FUNCTION_BLOCK EcMasterConfDevices IMPLEMENTS IEcTask
VAR_INPUT
END_VAR
VAR_OUTPUT
END_VAR
VAR
	iState : INT;
	masterConfDevices : Tc2_EtherCAT.FB_EcGetConfSlaves;
	_confDevices : ARRAY[0..Tc2_EtherCAT.EC_MAX_SLAVES] OF Tc2_EtherCAT.ST_EcSlaveConfigData;
	_execute: BOOL;
	_done: BOOL;
	_busy: BOOL;	
	_error: BOOL;
	_netId: AMSNETID;
END_VAR

CASE iState OF
	0:
		IF _execute THEN
			_done := FALSE;
			_busy := TRUE;
			_error := FALSE;
			masterConfDevices.bExecute := TRUE;
			IF masterConfDevices.bBusy THEN
				iState := 10;
				_execute := FALSE;
			END_IF
		END_IF
	10:
		IF NOT masterConfDevices.bBusy THEN
			IF NOT masterConfDevices.bError THEN
				_done := TRUE;
			ELSE
				_error := TRUE;
			END_IF
			_busy := FALSE;
			masterConfDevices.bExecute := FALSE;
			iState := 0;
		END_IF
END_CASE

masterConfDevices(sNetId := Tc2_System.F_CreateAmsNetId(nIds := NetId), 
					pArrEcConfSlaveInfo := ADR(_confDevices), 
					cbBufLen := SIZEOF(_confDevices));

{warning 'add method implementation '}
METHOD Abort : BOOL
masterConfDevices.bExecute := FALSE;
_busy := FALSE;
_execute := FALSE;
Abort := TRUE;
iState := 0;
END_METHOD

{warning 'add property implementation'}
PROPERTY Busy : BOOL
GET
Busy := _busy;
END_GET
END_PROPERTY

PROPERTY ConfiguredDevices : reference to array[0..Ec_Max_slaves] of St_ecslaveconfigdata
GET
ConfiguredDevices REF= _confDevices;
END_GET
END_PROPERTY

{warning 'add property implementation'}
PROPERTY Done : BOOL
GET
Done := _done;
END_GET
END_PROPERTY

{warning 'add property implementation'}
PROPERTY Error : BOOL
GET
Error := _error;
END_GET
END_PROPERTY

{warning 'add method implementation '}
METHOD Execute : BOOL
IF NOT masterConfDevices.bBusy THEN
	Execute := _execute := true;
END_IF
END_METHOD

{warning 'add property implementation'}
PROPERTY NetID : amsnetid
GET
NetID := _netId;
END_GET
SET
_netId := NetID;
END_SET
END_PROPERTY

PROPERTY NumberConfDevices : udint
GET
NumberConfDevices := masterConfDevices.nSlaves;
END_GET
END_PROPERTY

END_FUNCTION_BLOCK

(* stored: Version 1.1.0.1, ProductVersion 3.1.4024.11
   POU EcMasterConfDevices: Id {db18c880-11a0-493e-8ecc-75b7bb7d5ee1}, SpecialFunc None
   Method Abort: Id {29f4c6c7-c295-4b3b-88e0-1affbc2a49a0}
   Property Busy: Id {fbdf4132-a177-46bc-967b-0566d7f33115}
   Get Get: Id {5d58dddb-706d-4e38-b676-e06487ff79db}
   Property ConfiguredDevices: Id {fb01f319-f3bb-49a5-aaac-41e3704dce79}
   Get Get: Id {9f6170b9-866e-4cce-be3c-72b47ca25254}
   Property Done: Id {b48d60e5-568a-4737-82f5-f064f1fec13f}
   Get Get: Id {98963513-5a99-4ba5-9e68-de084642d9dc}
   Property Error: Id {26c57861-0c4e-4191-bdd5-0866724eb110}
   Get Get: Id {e6fa895d-b4d4-4640-9077-0f0f1302a60c}
   Method Execute: Id {f96e4b12-9f96-4f0d-b1b3-86c7ae262768}
   Property NetID: Id {be463b6e-fd1e-4a3e-a004-43e25ea0380d}
   Get Get: Id {b71f2620-a3b2-453b-be1a-abc40cfcb4c7}
   Set Set: Id {af88f21b-ce96-47c3-ae39-185f9073179e}
   Property NumberConfDevices: Id {4f2bd168-5a9c-426b-8942-886a695eff72}
   Get Get: Id {8c0a43a0-a55a-4b32-9366-54cb622486ca} *)
